{attribute 'qualified_only'}
VAR_GLOBAL
	
END_VAR

(* stored: Version 1.1.0.1, ProductVersion 3.1.4024.12
   GVL GVL_PROCESS: Id {bde269a9-07ec-44a2-b5d7-5697a0cb2c55} *)
